FUNCTION_BLOCK Rectangle (* openCV rectangle drawer *)
  (* Version 1.0, AN, SWDC RTSoft *)
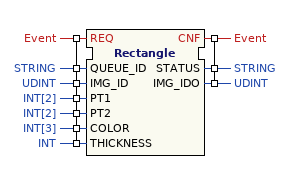
  EVENT_INPUT
    REQ WITH QUEUE_ID, IMG_ID, PT1, PT2, COLOR, THICKNESS;
  END_EVENT
  EVENT_OUTPUT
    CNF WITH STATUS, IMG_IDO;
  END_EVENT
  VAR_INPUT
    QUEUE_ID : STRING;
    IMG_ID : UDINT;
    PT1 : ARRAY [0..1] OF INT;
    PT2 : ARRAY [0..1] OF INT;
    COLOR : ARRAY [0..2] OF INT;
    THICKNESS : INT;
  END_VAR
  VAR_OUTPUT
    STATUS : STRING;
    IMG_IDO : UDINT;
  END_VAR
  ALGORITHM REQ IN ST:

  END_ALGORITHM
END_FUNCTION_BLOCK
